FUNCTION F_AdditionFunction : REAL
VAR_INPUT
	rInput1 : REAL;
	rInput2 : REAL;
END_VAR
VAR
END_VAR

F_AdditionFunction := rInput1 + rInput2;

END_FUNCTION

(* stored: Version 1.1.0.1, ProductVersion 3.1.4024.13
   POU F_AdditionFunction: Id {55b7c8b2-8888-4720-b92d-7d926238d4a7}, SpecialFunc None *)
